// TIA Portal V16 export
// export: Created 2022-02-04T14:40:20.1321727Z, ExportSetting WithDefaults, DisplayName Totally Integrated Automation Portal, DisplayVersion V16 Update 1, DisplayName TIA Portal Version Control Interface, DisplayVersion V16, DisplayName TIA Portal Openness, DisplayVersion V16, DisplayName SINAMICS Startdrive Advanced, DisplayVersion V16 Update 5, DisplayName SINAMICS Startdrive G130, G150, S120, S150, SINAMICS MV, S210, DisplayVersion V16 Update 5, DisplayName SINAMICS Startdrive G110M, G120, G120C, G120D, G120P, G115D, DisplayVersion V16 Update 5, DisplayName STEP 7 Professional, DisplayVersion V16, DisplayName STEP 7 Safety, DisplayVersion V16, DisplayName WinCC Advanced, DisplayVersion V16, DisplayName SIMATIC Visualization Architect, DisplayVersion V16
DATA_BLOCK "ServDB"   // DB5
VERSION : 0.1
// stored: AutoNumber true, InstanceOfName FB_Link_Server, InstanceOfType FB
"FB_Link_Server"
   // VAR RETAIN
   //    OperatorDetected : Bool;
   //    PackResortedReaded : Bool;
   //    FinishPackResorting : Bool;
   //    Enable2Sxema : Bool;
   //    EnableRolling : Bool;
   //    SettingsWasApplyied : Bool;
   //    CheckPlankL : Bool;
   //    FinishDefectPack : Bool;
   //    DefectPacketPushed : Bool;
   //    PackDefectReaded : Bool;
   //    PackParamChanged : Bool;
   //    PackReadyRidOff : Bool;
   //    GasketRidedOff : Bool;
   //    PackToPack : Bool;
   //    AddGasketLayer : Bool;
   //    PackBrakParamChanged : Bool;
   //    QPlankLayers : Int;
   //    VPlanksInPack : Int;
   //    QPlanksInLayer : Int;
   //    QPlanksInLayerBrak : Int;
   //    QPLankLayersBrak : Int;
   //    Sxema : DInt;
   //    SxemaNum : Int;
   //    PlankW : Int;
   //    PlankT : Int;
   //    Sxema2 : DInt;
   //    Sxema2Qlayers : Int;
   //    PackL : Int;
   //    PartId : DInt;
   //    PlankL : Int;
   //    ItemId : DInt;
   //    SetNumLayer : Int;
   //    SetNumPlankInLayer : Int;
   //    GeneralSpeed : Int;
   //    TotalPlanksInPack : Int;
   //    SetNumPlanksInLayerBrak : Int;
   //    CheckL : Int;
   //    GasketBrakPut : Bool;
   //    GasketLayersPeriod : Int;
   //    LineInWork : Bool;
   //    PackResorting : Bool;
   //    PackResorted : Bool;
   //    PackBrakComplete : Bool;
   //    RdyStartNewPack : Bool;
   //    RdyStart : Bool;
   //    DefectPacketResorted : Bool;
   //    NumLayerActual : Int;
   //    NumPlanksInLayerActual : Int;
   //    QPlanksOk : Int;
   //    QPlanksNotOk : Int;
   //    VPlanksOk : DInt;
   //    QPlankBrak : Int;
   //    VLayerOk : DInt;
   //    M_211 { S7_SetPoint := 'True'} : "ServIM";
   //    M_212 { S7_SetPoint := 'True'} : "ServIM";
   //    M_213 { S7_SetPoint := 'True'} : "ServIM";
   //    M_214 { S7_SetPoint := 'True'} : "ServIM";
   //    M_221 { S7_SetPoint := 'True'} : "ServIM";
   //    M_222 { S7_SetPoint := 'True'} : "ServIM";
   //    M_223 { S7_SetPoint := 'True'} : "ServIM";
   //    M_224 { S7_SetPoint := 'True'} : "ServIM";
   //    M_225 { S7_SetPoint := 'True'} : "ServIM";
   //    M_231 { S7_SetPoint := 'True'} : "ServIM";
   //    M_232 { S7_SetPoint := 'True'} : "ServIM";
   //    M_233 { S7_SetPoint := 'True'} : "ServIM";
   //    ForkRotator { S7_SetPoint := 'True'} : "ServIM";
   //    M_234 { S7_SetPoint := 'True'} : "ServIM";
   //    M_235 { S7_SetPoint := 'True'} : "ServIM";
   //    M_311 { S7_SetPoint := 'True'} : "ServIM";
   //    M_312 { S7_SetPoint := 'True'} : "ServIM";
   //    M_313 { S7_SetPoint := 'True'} : "ServIM";
   //    M_314 { S7_SetPoint := 'True'} : "ServIM";
   //    M_315 { S7_SetPoint := 'True'} : "ServIM";
   //    M_316 { S7_SetPoint := 'True'} : "ServIM";
   //    M_317 { S7_SetPoint := 'True'} : "ServIM";
   //    GasketSupplier { S7_SetPoint := 'True'} : "ServIM";
   //    M_321 { S7_SetPoint := 'True'} : "ServIM";
   //    M_322 { S7_SetPoint := 'True'} : "ServIM";
   //    M_323 { S7_SetPoint := 'True'} : "ServIM";
   //    M_324 { S7_SetPoint := 'True'} : "ServIM";
   //    M_325 { S7_SetPoint := 'True'} : "ServIM";
   //    M_330 { S7_SetPoint := 'True'} : "ServIM";
   //    M_331 { S7_SetPoint := 'True'} : "ServIM";
   //    M_332 { S7_SetPoint := 'True'} : "ServIM";
   //    M_333 { S7_SetPoint := 'True'} : "ServIM";
   //    M_334 { S7_SetPoint := 'True'} : "ServIM";
   //    M_335 { S7_SetPoint := 'True'} : "ServIM";
   //    M_336 { S7_SetPoint := 'True'} : "ServIM";
   //    Alarm_List { S7_SetPoint := 'True'} : Array[0..255] of Bool;
   // END_VAR
BEGIN
END_DATA_BLOCK
